// TIA Portal V20 export
TYPE "TypeIOLinkParamArray"
   STRUCT
      Param { ExternalAccessible := 'False'; ExternalVisible := 'False'; ExternalWritable := 'False'} : Array[0..9] of "TypeIOLinkParam";
   END_STRUCT;
END_TYPE
